PROGRAM Production_00
VAR
i : INT;
END_VAR


// write production line commands (from visu) down to each units pack tags

FOR i := 1 TO 4 DO
	GVL.UnitPackTags[i] :=  GVL.LineCommands;
END_FOR

END_PROGRAM

(* stored: Version 1.1.0.1, ProductVersion 3.1.4024.11
   POU Production_00: Id {5dc5c6b7-6f8e-4f7c-94a8-20d2f19a34d3}, SpecialFunc None *)
